FUNCTION_BLOCK UPDATE_CONV_STATE (* Composite Function Block Type *)
  (* Standard: 61499-2 *)
  (* Version 0.2, 2003-12-05, JHC, Rockwell Automation, Renamed from NEWCOMPFB. *)
  (* Version 0.1, 2002-01-08, JHC, Rockwell Automation, Added DLY FB as example. *)
  (* Version 0.0, 2000-05-27, JHC, Rockwell Automation *)
  (* Compiler header: package fb.rt.template; *)
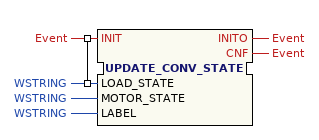
  EVENT_INPUT
    INIT WITH LOAD_STATE; (* Initialization Request *)
  END_EVENT
  EVENT_OUTPUT
    INITO; (* Initialization Confirm *)
    CNF; (* Execution Confirmation *)
  END_EVENT
  VAR_INPUT
    LOAD_STATE : WSTRING; (* Input event qualifier *)
    MOTOR_STATE : WSTRING;
    LABEL : WSTRING;
  END_VAR
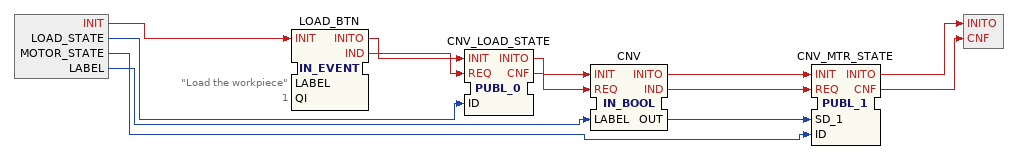
  FBS
    LOAD_BTN : IN_EVENT(LABEL := "Load the workpiece", QI := 1);
    CNV_LOAD_STATE : PUBL_0;
    CNV : IN_BOOL;
    CNV_MTR_STATE : PUBL_1;
  END_FBS
  EVENT_CONNECTIONS
    LOAD_BTN.INITO TO CNV_LOAD_STATE.INIT;
    CNV_LOAD_STATE.INITO TO CNV.INIT;
    CNV.INITO TO CNV_MTR_STATE.INIT;
    INIT TO LOAD_BTN.INIT;
    LOAD_BTN.IND TO CNV_LOAD_STATE.REQ;
    CNV_LOAD_STATE.CNF TO CNV.REQ;
    CNV.IND TO CNV_MTR_STATE.REQ;
    CNV_MTR_STATE.INITO TO INITO;
    CNV_MTR_STATE.CNF TO CNF;
  END_CONNECTIONS
  DATA_CONNECTIONS
    CNV.OUT TO CNV_MTR_STATE.SD_1;
    LOAD_STATE TO CNV_LOAD_STATE.ID;
    LABEL TO CNV.LABEL;
    MOTOR_STATE TO CNV_MTR_STATE.ID;
  END_CONNECTIONS
END_FUNCTION_BLOCK
